FUNCTION_BLOCK Q_LineAttributes (* Command change line attributes ( Part 6 - F.30 ) *)
  (* Standard: ISO 11783-6; Description: This command is used to change the line attributes in a line attributes object. Return values iso_s16 - E_NO_ERR - OK - E_OVERFLOW - buffer overflow - E_NOACT - Command not possible in current state - E_NO_INSTANCE - No VT client available *)
  (* Version 1.0, 2022-07-08, franz *)
  (* Documentation:
  This command is used to change the line attributes in a line attributes object.
   Return values
   iso_s16
    - E_NO_ERR - OK
   - E_OVERFLOW - buffer overflow
   - E_NOACT - Command not possible in current state
   - E_NO_INSTANCE - No VT client available
  *)
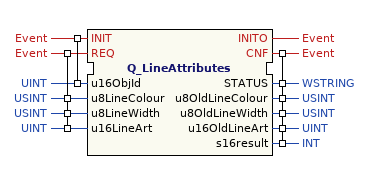
  EVENT_INPUT
    INIT WITH u16ObjId; (* Service Initialization *)
    REQ WITH u8LineColour, u8LineWidth, u16LineArt; (* Service Request *)
  END_EVENT
  EVENT_OUTPUT
    INITO; (* Initialization Confirm *)
    CNF WITH STATUS, s16result, u8OldLineColour, u8OldLineWidth, u16OldLineArt; (* Confirmation of Requested Service *)
  END_EVENT
  VAR_INPUT
    u16ObjId : UINT; (* Object ID *)
    u8LineColour : USINT; (* New line colour *)
    u8LineWidth : USINT; (* New line width (see Part 6 - B.14.3) *)
    u16LineArt : UINT; (* New line art (see Part 6 - B.14.3) *)
  END_VAR
  VAR_OUTPUT
    STATUS : WSTRING; (* Service Status *)
    u8OldLineColour : USINT; (* Old line colour *)
    u8OldLineWidth : USINT; (* Old line width (see Part 6 - B.14.3) *)
    u16OldLineArt : UINT; (* Old line art (see Part 6 - B.14.3) *)
    s16result : INT; (* retval see description *)
  END_VAR
END_FUNCTION_BLOCK
